// TIA Portal V19 export
TYPE "TExtEncoder_ErrorWord"
// stored: Access Published
   STRUCT
      SystemFault : Bool;
      ConfigFault : Bool;
      UserFault : Bool;
      CommandNotAccepted : Bool;
      SensorFault : Bool;
      CommunicationFault : Bool;
      HomingError : Bool;
      PeripheralError : Bool;
   END_STRUCT;
END_TYPE
